FUNCTION_BLOCK FB_ReceipeList
VAR_INPUT
	sReceipeListIn			:STRING(1000);
END_VAR
VAR_OUTPUT
	sReceipeListOut			:STRING(1000);
	sReceipe				:STRING;
	bEmpty					:BOOL;
END_VAR
VAR
	nPosition				:INT;
END_VAR

nPosition := FIND(sReceipeListIn,';');
IF nPosition > 0 THEN
	sReceipe := LEFT(sReceipeListIn,(nPosition - 1));
	sReceipeListOut	:= DELETE(sReceipeListIn,(nPosition + 1),0);
ELSE
	sReceipe := sReceipeListIn;
	sReceipeListOut	:= '';
END_IF
bEmpty := (LEN(sReceipeListOut) <= 0);

END_FUNCTION_BLOCK

(* stored: Version 1.1.0.1, ProductVersion 3.1.4024.10
   POU FB_ReceipeList: Id {16d70c4a-aa1f-417f-a9ec-c697a66b5478}, SpecialFunc None *)
